// TIA Portal project "parking_lot" (V15.1)

(* hardware
DEVICE "S7-1200 station_1"  S7-1200 Station
   slot 0: "Rack_0"  S7-1200 Rack  Rack  V1.0
   slot 1: "PLC_1"  CPU 1215C DC/DC/DC  6ES7 215-1AG40-0XB0  V4.2
*)

// ===== PLC "PLC_1"  CPU 1215C DC/DC/DC =====

VAR_GLOBAL   // PLC tag table "Default tag table"
   "start" AT %I0.0 : Bool;
   "stop" AT %I0.1 : Bool;
   "mem_1" AT %M0.0 : Bool;
   "ent_sensor" AT %M0.1 : Bool;
   "out_sensor" AT %M0.2 : Bool;
   "green" AT %Q0.0 : Bool;
   "yellow" AT %Q0.1 : Bool;
   "red" AT %Q0.2 : Bool;
   "Tag_1" AT %MD200 : Time;
   "reset" AT %I0.2 : Bool;
   "Tag_2" AT %MW500 : Int;
   "Tag_3" AT %Q0.3 : Bool;
   "clock" AT %M1.7 : Bool;
   "Clock_Byte" AT %MB1 : Byte;
   "Clock_10Hz" AT %M1.0 : Bool;
   "Clock_5Hz" AT %M1.1 : Bool;
   "Clock_2.5Hz" AT %M1.2 : Bool;
   "Clock_2Hz" AT %M1.3 : Bool;
   "Clock_1.25Hz" AT %M1.4 : Bool;
   "Clock_1Hz" AT %M1.5 : Bool;
   "Clock_0.625Hz" AT %M1.6 : Bool;
   "Clock_0.5Hz" AT %M1.7 : Bool;
END_VAR

// folder: System blocks/Program resources

DATA_BLOCK "Car_Counter"   // DB2
{ S7_Optimized_Access := 'TRUE' }
AUTHOR : Simatic
FAMILY : IEC
NAME : CNTR
VERSION : 1.0
// stored: InstanceOfName IEC_COUNTER
"IEC_COUNTER"
BEGIN
END_DATA_BLOCK

// folder: (top level)

ORGANIZATION_BLOCK "Main"   // OB1, LAD, ProgramCycle
TITLE = "Main Program Sweep (Cycle)"
{ S7_Optimized_Access := 'TRUE' }
VERSION : 0.1
   VAR_INPUT
      Initial_Call : Bool;   // Initial call of this OB
      Remanence : Bool;   // =True, if remanent data are available
   END_VAR
BEGIN

REGION Network 1
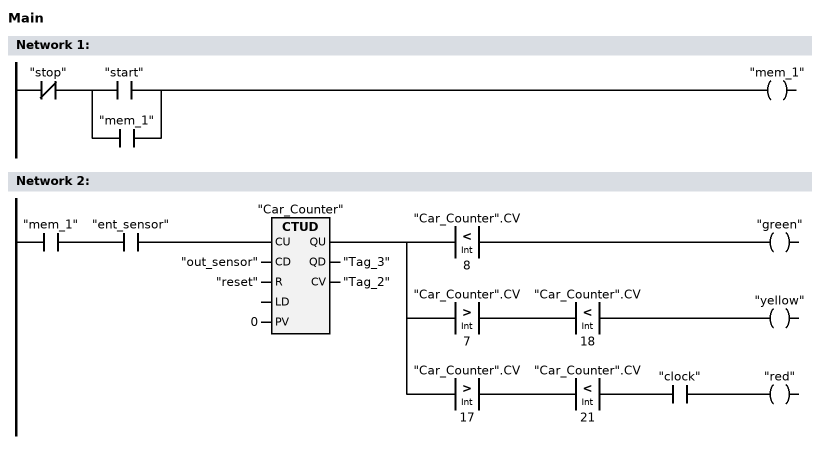
   RUNG wire#powerrail
      I_Contact( "stop" )
      wire#w1
      Contact( "start" )
      wire#w2
      Coil( "mem_1" )
   END_RUNG
   RUNG wire#w1
      Contact( "mem_1" )
   END_RUNG wire#w2
   // the same network as SCL:
   "mem_1" := NOT "stop" AND ("start" OR "mem_1");
END_REGION

REGION Network 2
   "Car_Counter".CTUD(CU := "mem_1" AND "ent_sensor",
                      CD := "out_sensor",
                      R := "reset",
                      PV := 0,
                      QD => "Tag_3",
                      CV => "Tag_2");
   "green" := "Car_Counter".QU AND ("Car_Counter".CV < 8);
   "yellow" := "Car_Counter".QU AND ("Car_Counter".CV > 7) AND ("Car_Counter".CV < 18);
   "red" := "Car_Counter".QU AND ("Car_Counter".CV > 17) AND ("Car_Counter".CV < 21) AND "clock";
END_REGION
END_ORGANIZATION_BLOCK